{attribute addProperty BoxType "EL3403-0000-0017"}
{attribute addProperty Id "Sync_ErrorAT %I*BOOL8114TxPDO_ToggleAT %I*BOOL819CurrentAT %I*DINT32417VoltageAT %I*DINT32418Active_powerAT %I*DINT32419IndexAT %I*USINT8120VariantValueAT %I*DINT32429"}
{attribute addProperty CRC "4279382388"}
{attribute addProperty SizeInBites "152"}
{attribute addProperty SizeInBytes "19"}
TYPE PM_Inputs_Channel_FF123174 :
STRUCT
	{attribute addProperty Name "Sync_Error"}
	Sync_Error AT %I* : BOOL;
	{attribute addProperty Name "TxPDO_Toggle"}
	TxPDO_Toggle AT %I* : BOOL;
	{attribute addProperty Name "Current"}
	Current AT %I* : DINT;
	{attribute addProperty Name "Voltage"}
	Voltage AT %I* : DINT;
	{attribute addProperty Name "Active_power"}
	Active_power AT %I* : DINT;
	{attribute addProperty Name "Index"}
	Index AT %I* : USINT;
	{attribute addProperty Name "VariantValue"}
	VariantValue AT %I* : DINT;
END_STRUCT
END_TYPE

(* stored: Version 1.2.0.0, ProductVersion 3.1.4024.9
   DUT PM_Inputs_Channel_FF123174: Id {eaf07062-eb7f-4e00-92d1-253d81c6cfc0} *)
